# EPICS autosave request: soft_iocs/meas_comp/iocBoot/iocmeas_comp_ctr/dark.req
file "ao.req", P=$(P)Dark, R=1
file "ao.req", P=$(P)Dark, R=2
file "ao.req", P=$(P)Dark, R=3
file "ao.req", P=$(P)Dark, R=4
file "ao.req", P=$(P)Dark, R=5
file "ao.req", P=$(P)Dark, R=6
file "ao.req", P=$(P)Dark, R=7
file "ao.req", P=$(P)Dark, R=8
